INTERFACE ITF_Component_TE1_HMI_Connector EXTENDS ITF_BaseComponent_HMI_Connector

END_INTERFACE

(* stored: Version 1.1.0.1, ProductVersion 3.1.4024.15
   Itf ITF_Component_TE1_HMI_Connector: Id {826cb8fa-9974-4613-ad75-6bce6db69f8f} *)
